// Mitsubishi GX Works2 project: 12   PLC: FX2N/FX2NC

PROGRAM MAIN
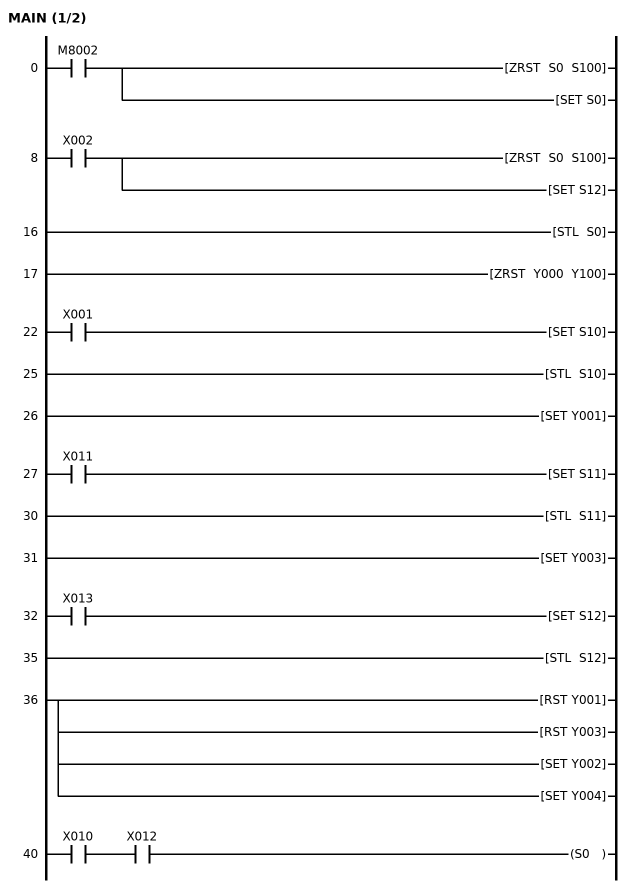
0     LD      M8002
      ZRST    S0 S100
      SET     S0
8     LD      X002
      ZRST    S0 S100
      SET     S12
16    STL     S0
17    ZRST    Y000 Y100
22    LD      X001
      SET     S10
25    STL     S10
26    SET     Y001
27    LD      X011
      SET     S11
30    STL     S11
31    SET     Y003
32    LD      X013
      SET     S12
35    STL     S12
36    RST     Y001
      RST     Y003
      SET     Y002
      SET     Y004
40    LD      X010
      AND     X012
      OUT     S0
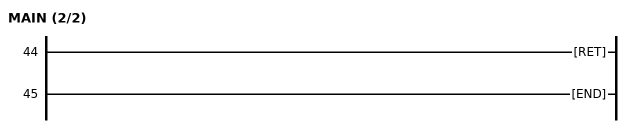
44    RET
45    END
END_PROGRAM

// device comments not shown above
BL0  ; main
BL1  ; a
BL2  ; b
